Omron CX-Programmer project NewProject (CX-Programmer 9.03)

# PLC CLP: CJ1M CPU11
I/O table (CPU CJ1M-CPU11): rack 0 slot 0 CJ1W-ETN21(ETN11Mode); rack 0 slot 1 CJ1W-ID211; rack 0 slot 2 CJ1W-OD211; rack 0 slot 3 CJ1W-ID211; rack 0 slot 4 CJ1W-OD211; rack 0 slot 5 CJ1W-ID211; rack 0 slot 6 CJ1W-OD232

## Program Armazem (cyclic task 0)
Local symbols
AS_RS_Ativado 5.02 BOOL
AUX_CTRG W10.02 BOOL
AUX_X_OK W10.05 BOOL
AUX_Y_OK W10.07 BOOL
AUX_Z_OK W10.06 BOOL
Confirmacao W4.00 BOOL
Eletroval1 1.06 BOOL
Eletroval2 1.07 BOOL
Eletroval3 1.08 BOOL
Eletroval4 1.09 BOOL
Elevar_Z W15.00 BOOL
Esteira1 1.00 BOOL
Esteira2 1.01 BOOL
Esteira3 1.02 BOOL
Esteira4 1.03 BOOL
Etapa BOOL
Etapa0 W0.00 BOOL
Etapa1 W0.01 BOOL
Etapa10 W1.02 BOOL
Etapa11 W1.03 BOOL
Etapa2 W0.02 BOOL
Etapa3 W0.03 BOOL
Etapa4 W0.04 BOOL
Etapa5 W0.05 BOOL
Etapa6 W0.06 BOOL
Etapa7 W0.07 BOOL
Etapa8 W1.00 BOOL
Etapa9 W1.01 BOOL
Home_X_Completo 4.05 BOOL
Home_Y_Completo 4.07 BOOL
Home_Z_Completo 4.09 BOOL
Pos_X_Completa 4.04 BOOL
Pos_Y_Completa 4.06 BOOL
Pos_Z_Completa 4.08 BOOL
Sensor1 0.00 BOOL
Sensor2 0.01 BOOL
Sensor3 0.02 BOOL
Sensor4 0.03 BOOL
X_CTRG 5.04 BOOL
X_D0 5.05 BOOL
X_D1 5.06 BOOL
X_D2 5.07 BOOL
X_D3 5.08 BOOL
X_To_Home 5.03 BOOL
Y_CTRG 5.10 BOOL
Y_D0 5.11 BOOL
Y_D1 5.12 BOOL
Y_D2 5.13 BOOL
Y_D3 5.14 BOOL
Y_To_Home 5.09 BOOL
Z_CTRG 6.00 BOOL
Z_D0 6.01 BOOL
Z_D1 6.02 BOOL
Z_D2 6.03 BOOL
Z_D3 6.04 BOOL
Z_To_Home 5.15 BOOL
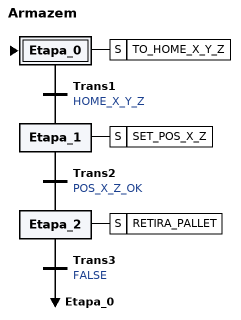
INITIAL_STEP Etapa_0 :
TO_HOME_X_Y_Z(S) ;
END_STEP
TRANSITION Trans1 FROM Etapa_0 TO Etapa_1
 := HOME_X_Y_Z;
END_TRANSITION
STEP Etapa_1 :
SET_POS_X_Z(S) ;
END_STEP
TRANSITION Trans2 FROM Etapa_1 TO Etapa_2
 := POS_X_Z_OK;
END_TRANSITION
STEP Etapa_2 :
RETIRA_PALLET(S) ;
END_STEP
TRANSITION Trans3 FROM Etapa_2 TO Etapa_0
 := FALSE;
END_TRANSITION

### Action TO_HOME_X_Y_Z

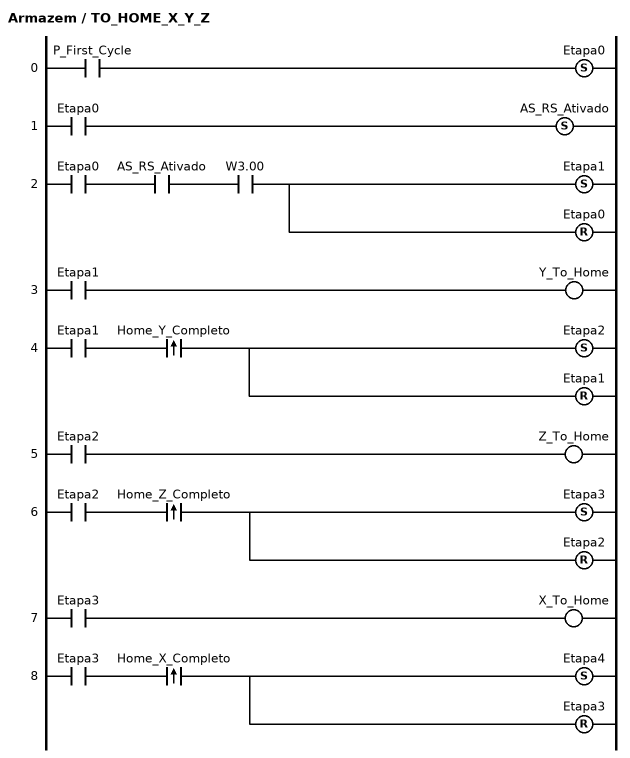
; rung 0
LD P_First_Cycle
SET Etapa0
; rung 1
LD Etapa0
SET AS_RS_Ativado
; rung 2
LD Etapa0
AND AS_RS_Ativado
AND W3.00
SET Etapa1
RSET Etapa0
; rung 3
LD Etapa1
OUT Y_To_Home
; rung 4
LD Etapa1
@AND Home_Y_Completo
SET Etapa2
RSET Etapa1
; rung 5
LD Etapa2
OUT Z_To_Home
; rung 6
LD Etapa2
@AND Home_Z_Completo
SET Etapa3
RSET Etapa2
; rung 7
LD Etapa3
OUT X_To_Home
; rung 8
LD Etapa3
@AND Home_X_Completo
SET Etapa4
RSET Etapa3

### Action SET_POS_X_Z

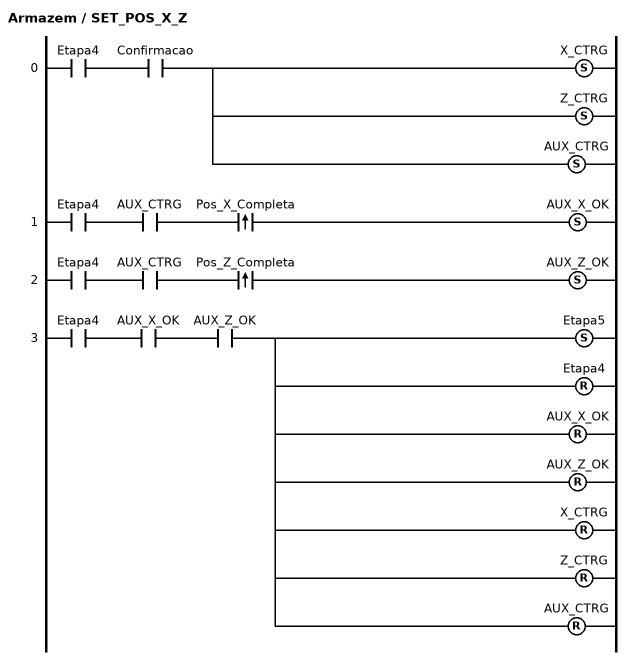
; rung 0
LD Etapa4
AND Confirmacao
SET X_CTRG
SET Z_CTRG
SET AUX_CTRG
; rung 1
LD Etapa4
AND AUX_CTRG
@AND Pos_X_Completa
SET AUX_X_OK
; rung 2
LD Etapa4
AND AUX_CTRG
@AND Pos_Z_Completa
SET AUX_Z_OK
; rung 3
LD Etapa4
AND AUX_X_OK
AND AUX_Z_OK
SET Etapa5
RSET Etapa4
RSET AUX_X_OK
RSET AUX_Z_OK
RSET X_CTRG
RSET Z_CTRG
RSET AUX_CTRG

### Action RETIRA_PALLET

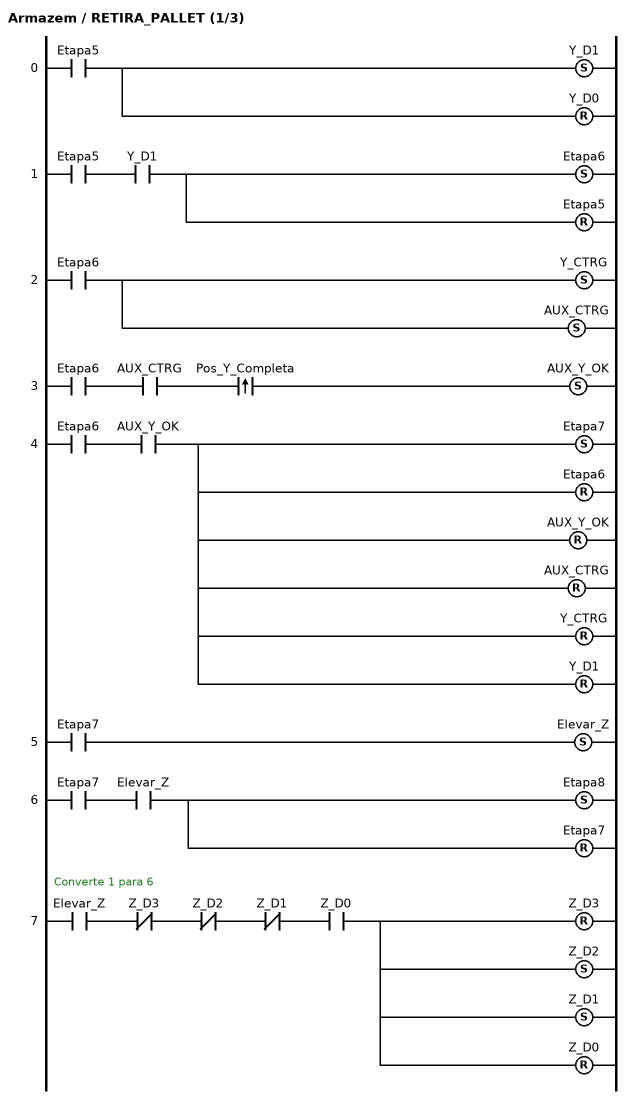
; rung 0
LD Etapa5
SET Y_D1
RSET Y_D0
; rung 1
LD Etapa5
AND Y_D1
SET Etapa6
RSET Etapa5
; rung 2
LD Etapa6
SET Y_CTRG
SET AUX_CTRG
; rung 3
LD Etapa6
AND AUX_CTRG
@AND Pos_Y_Completa
SET AUX_Y_OK
; rung 4
LD Etapa6
AND AUX_Y_OK
SET Etapa7
RSET Etapa6
RSET AUX_Y_OK
RSET AUX_CTRG
RSET Y_CTRG
RSET Y_D1
; rung 5
LD Etapa7
SET Elevar_Z
; rung 6
LD Etapa7
AND Elevar_Z
SET Etapa8
RSET Etapa7
; rung 7: Converte 1 para 6
LD Elevar_Z
ANDNOT Z_D3
ANDNOT Z_D2
ANDNOT Z_D1
AND Z_D0
RSET Z_D3
SET Z_D2
SET Z_D1
RSET Z_D0

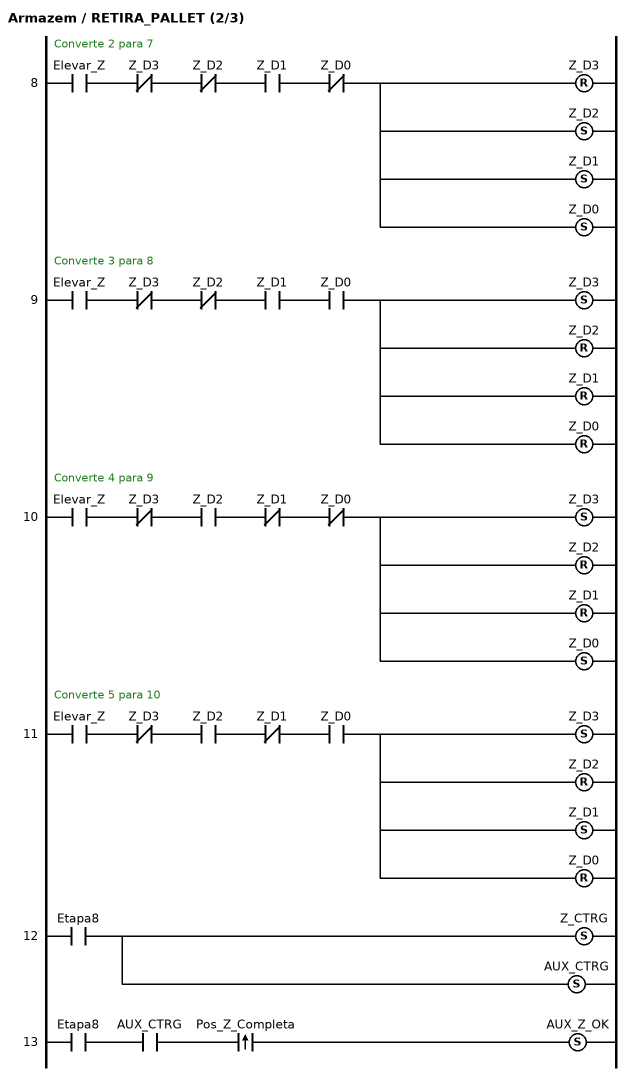
; rung 8: Converte 2 para 7
LD Elevar_Z
ANDNOT Z_D3
ANDNOT Z_D2
AND Z_D1
ANDNOT Z_D0
RSET Z_D3
SET Z_D2
SET Z_D1
SET Z_D0
; rung 9: Converte 3 para 8
LD Elevar_Z
ANDNOT Z_D3
ANDNOT Z_D2
AND Z_D1
AND Z_D0
SET Z_D3
RSET Z_D2
RSET Z_D1
RSET Z_D0
; rung 10: Converte 4 para 9
LD Elevar_Z
ANDNOT Z_D3
AND Z_D2
ANDNOT Z_D1
ANDNOT Z_D0
SET Z_D3
RSET Z_D2
RSET Z_D1
SET Z_D0
; rung 11: Converte 5 para 10
LD Elevar_Z
ANDNOT Z_D3
AND Z_D2
ANDNOT Z_D1
AND Z_D0
SET Z_D3
RSET Z_D2
SET Z_D1
RSET Z_D0
; rung 12
LD Etapa8
SET Z_CTRG
SET AUX_CTRG
; rung 13
LD Etapa8
AND AUX_CTRG
@AND Pos_Z_Completa
SET AUX_Z_OK

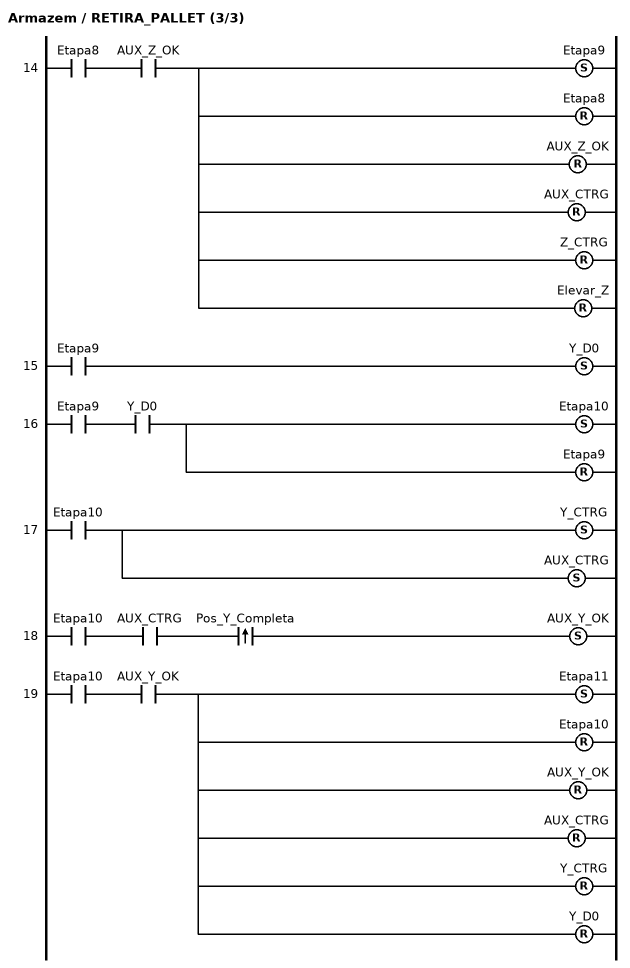
; rung 14
LD Etapa8
AND AUX_Z_OK
SET Etapa9
RSET Etapa8
RSET AUX_Z_OK
RSET AUX_CTRG
RSET Z_CTRG
RSET Elevar_Z
; rung 15
LD Etapa9
SET Y_D0
; rung 16
LD Etapa9
AND Y_D0
SET Etapa10
RSET Etapa9
; rung 17
LD Etapa10
SET Y_CTRG
SET AUX_CTRG
; rung 18
LD Etapa10
AND AUX_CTRG
@AND Pos_Y_Completa
SET AUX_Y_OK
; rung 19
LD Etapa10
AND AUX_Y_OK
SET Etapa11
RSET Etapa10
RSET AUX_Y_OK
RSET AUX_CTRG
RSET Y_CTRG
RSET Y_D0

### Transition HOME_X_Y_Z
; HOME_OK(X, Y, Z)

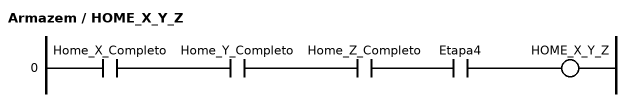
; rung 0
LD Home_X_Completo
AND Home_Y_Completo
AND Home_Z_Completo
AND Etapa4
OUT HOME_X_Y_Z

### Transition POS_X_Z_OK

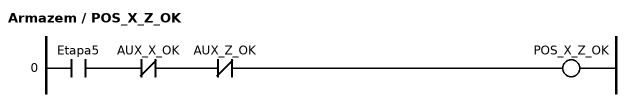
; rung 0
LD Etapa5
ANDNOT AUX_X_OK
ANDNOT AUX_Z_OK
OUT POS_X_Z_OK

## Program NewProgram1 (cyclic task 0)
Local symbols
AS_RS_Ativado 5.02 BOOL
AS_RS_Eixo_X_Ctrg 5.04 BOOL
AS_RS_Eixo_X_D0 5.05 BOOL
AS_RS_Eixo_X_D1 5.06 BOOL
AS_RS_Eixo_X_D2 5.07 BOOL
AS_RS_Eixo_X_D3 5.08 BOOL
AS_RS_Eixo_X_To_Home 5.03 BOOL
AS_RS_Eixo_Y_Ctrg 5.10 BOOL
AS_RS_Eixo_Y_D0 5.11 BOOL
AS_RS_Eixo_Y_D1 5.12 BOOL
AS_RS_Eixo_Y_D2 5.13 BOOL
AS_RS_Eixo_Y_D3 5.14 BOOL
AS_RS_Eixo_Y_To_Home 5.09 BOOL
AS_RS_Eixo_Z_Ctrg 6.00 BOOL
AS_RS_Eixo_Z_D0 6.01 BOOL
AS_RS_Eixo_Z_D1 6.02 BOOL
AS_RS_Eixo_Z_D2 6.03 BOOL
AS_RS_Eixo_Z_D3 6.04 BOOL
AS_RS_Eixo_Z_To_Home 5.15 BOOL
AS_RS_Home_X_Completo 4.05 BOOL
AS_RS_Home_Y_Completo 4.07 BOOL
AS_RS_Home_Z_Completo 4.09 BOOL
AS_RS_Pos_X_Completa 4.04 BOOL
AS_RS_Pos_Y_Completa 4.06 BOOL
AS_RS_Pos_Z_Completa 4.08 BOOL
Confirmacao W4.00 BOOL
Eletroval1 1.06 BOOL
Eletroval2 1.07 BOOL
Eletroval3 1.08 BOOL
Eletroval4 1.09 BOOL
Esteira1 1.00 BOOL
Esteira2 1.01 BOOL
Esteira3 1.02 BOOL
Esteira4 1.03 BOOL
Etapa BOOL
Etapa0 W0.00 BOOL
Etapa1 W0.01 BOOL
Etapa10 W1.02 BOOL
Etapa11 W1.03 BOOL
Etapa2 W0.02 BOOL
Etapa3 W0.03 BOOL
Etapa4 W0.04 BOOL
Etapa5 W0.05 BOOL
Etapa6 W0.06 BOOL
Etapa7 W0.07 BOOL
Etapa8 W1.00 BOOL
Etapa9 W1.01 BOOL
Sensor1 0.00 BOOL
Sensor2 0.01 BOOL
Sensor3 0.02 BOOL
Sensor4 0.03 BOOL

### Section Main

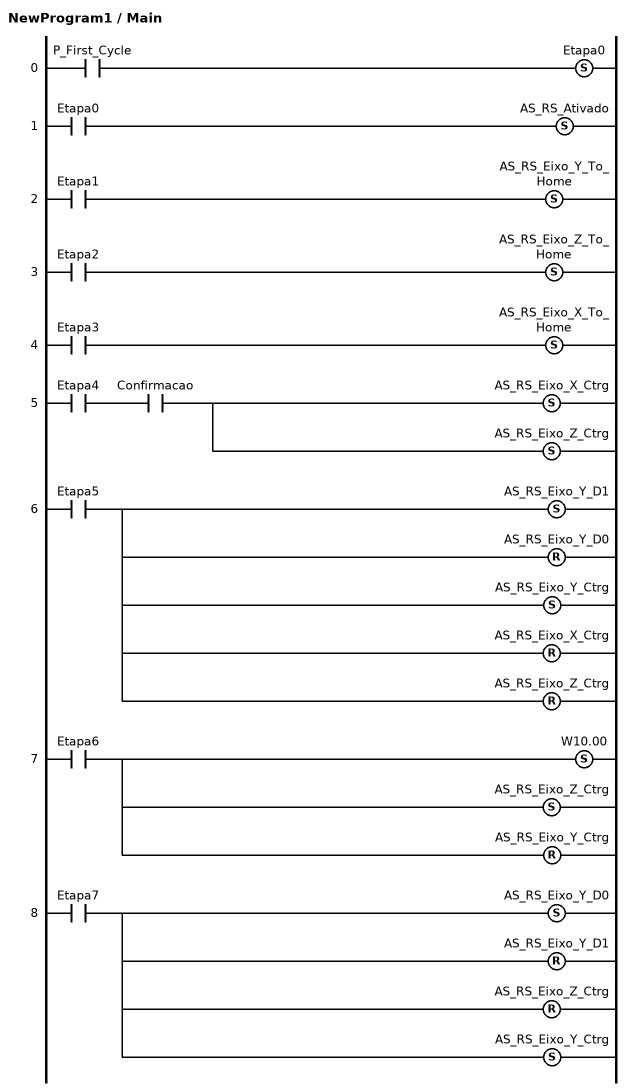
; rung 0
LD P_First_Cycle
SET Etapa0
; rung 1
LD Etapa0
SET AS_RS_Ativado
; rung 2
LD Etapa1
SET AS_RS_Eixo_Y_To_Home
; rung 3
LD Etapa2
SET AS_RS_Eixo_Z_To_Home
; rung 4
LD Etapa3
SET AS_RS_Eixo_X_To_Home
; rung 5
LD Etapa4
AND Confirmacao
SET AS_RS_Eixo_X_Ctrg
SET AS_RS_Eixo_Z_Ctrg
; rung 6
LD Etapa5
SET AS_RS_Eixo_Y_D1
RSET AS_RS_Eixo_Y_D0
SET AS_RS_Eixo_Y_Ctrg
RSET AS_RS_Eixo_X_Ctrg
RSET AS_RS_Eixo_Z_Ctrg
; rung 7
LD Etapa6
SET W10.00
SET AS_RS_Eixo_Z_Ctrg
RSET AS_RS_Eixo_Y_Ctrg
; rung 8
LD Etapa7
SET AS_RS_Eixo_Y_D0
RSET AS_RS_Eixo_Y_D1
RSET AS_RS_Eixo_Z_Ctrg
SET AS_RS_Eixo_Y_Ctrg

### Section Transitions

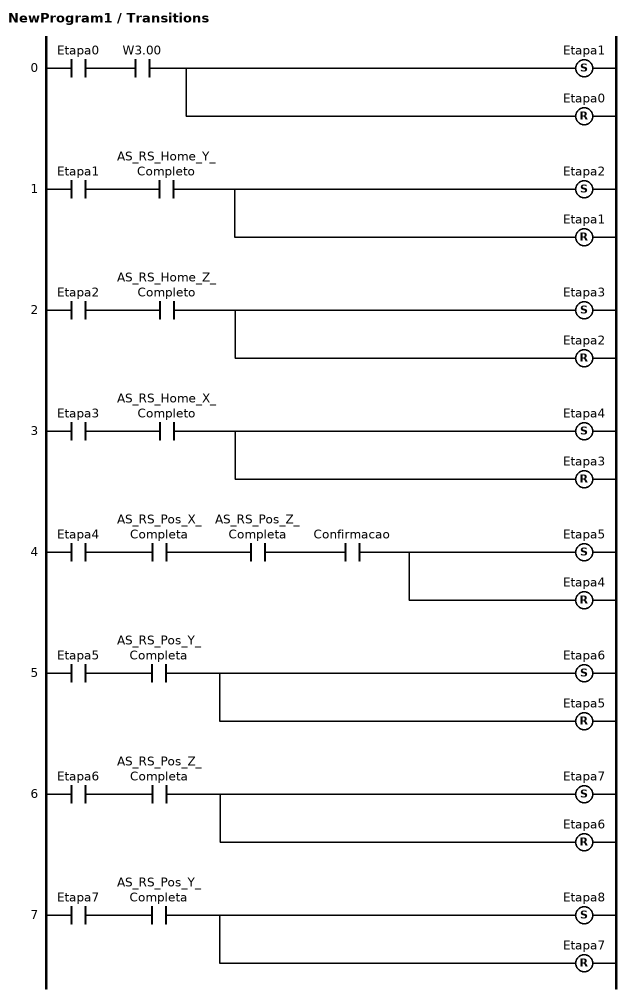
; rung 0
LD Etapa0
AND W3.00
SET Etapa1
RSET Etapa0
; rung 1
LD Etapa1
AND AS_RS_Home_Y_Completo
SET Etapa2
RSET Etapa1
; rung 2
LD Etapa2
AND AS_RS_Home_Z_Completo
SET Etapa3
RSET Etapa2
; rung 3
LD Etapa3
AND AS_RS_Home_X_Completo
SET Etapa4
RSET Etapa3
; rung 4
LD Etapa4
AND AS_RS_Pos_X_Completa
AND AS_RS_Pos_Z_Completa
AND Confirmacao
SET Etapa5
RSET Etapa4
; rung 5
LD Etapa5
AND AS_RS_Pos_Y_Completa
SET Etapa6
RSET Etapa5
; rung 6
LD Etapa6
AND AS_RS_Pos_Z_Completa
SET Etapa7
RSET Etapa6
; rung 7
LD Etapa7
AND AS_RS_Pos_Y_Completa
SET Etapa8
RSET Etapa7

### Section END
; rung 0
END(001)